(* IEC 61131-3 sources: BnR-PLC-motor-configuration/ncsdcctrl, 3 files *)

(* ---- ncsdcctrl.var ---- *)
VAR
	gAxis01_oSetPosOld : INT := 0;
	gAxis02_oSetPosOld : INT := 0;
	gAxis03_oSetPosOld : INT := 0;
END_VAR

(* ---- ncsdcctrlCyclic.st ---- *)
PROGRAM _CYCLIC

(* ### BEGIN gAxis01 ### *)

(* life counter emulation of digital inputs *)
      gAxis01_DiDoIf.iLifeCntReference := gAxis01_DiDoIf.iLifeCntReference + 1;
      gAxis01_DiDoIf.iLifeCntNegHwEnd  := gAxis01_DiDoIf.iLifeCntNegHwEnd  + 1;
      gAxis01_DiDoIf.iLifeCntPosHwEnd  := gAxis01_DiDoIf.iLifeCntPosHwEnd  + 1;

(* default function model of ACOPOSmicro: convert absolute steps to delta steps - overflow save delta calculation *)
      gAxis01_MotorStep0 := gAxis01_DrvIf.oSetPos - gAxis01_oSetPosOld;
      gAxis01_oSetPosOld := gAxis01_DrvIf.oSetPos;

(* ### END gAxis01 ### *)

(* ### BEGIN gAxis02 ### *)

(* life counter emulation of digital inputs *)
      gAxis02_DiDoIf.iLifeCntReference := gAxis02_DiDoIf.iLifeCntReference + 1;
      gAxis02_DiDoIf.iLifeCntNegHwEnd  := gAxis02_DiDoIf.iLifeCntNegHwEnd  + 1;
      gAxis02_DiDoIf.iLifeCntPosHwEnd  := gAxis02_DiDoIf.iLifeCntPosHwEnd  + 1;

(* default function model of ACOPOSmicro: convert absolute steps to delta steps - overflow save delta calculation *)
      gAxis02_MotorStep0 := gAxis02_DrvIf.oSetPos - gAxis02_oSetPosOld;
      gAxis02_oSetPosOld := gAxis02_DrvIf.oSetPos;

(* ### END gAxis02 ### *)

(* ### BEGIN gAxis03 ### *)

(* life counter emulation of digital inputs *)
      gAxis03_DiDoIf.iLifeCntReference := gAxis03_DiDoIf.iLifeCntReference + 1;
      gAxis03_DiDoIf.iLifeCntNegHwEnd  := gAxis03_DiDoIf.iLifeCntNegHwEnd  + 1;
      gAxis03_DiDoIf.iLifeCntPosHwEnd  := gAxis03_DiDoIf.iLifeCntPosHwEnd  + 1;

(* default function model of ACOPOSmicro: convert absolute steps to delta steps - overflow save delta calculation *)
      gAxis03_MotorStep0 := gAxis03_DrvIf.oSetPos - gAxis03_oSetPosOld;
      gAxis03_oSetPosOld := gAxis03_DrvIf.oSetPos;

(* ### END gAxis03 ### *)

END_PROGRAM

(* ---- ncsdcctrlInit.st ---- *)
PROGRAM _INIT

(* ### BEGIN gAxis01 ### *)

(* initialize general interfaces *)
      gAxis01.size := gAxis01.size;
      gAxis01_HW.DrvIf_Typ := ncSDC_DRVSM16;
      brsstrcpy( ADR(gAxis01_HW.DrvIf_Name[0]), ADR('gAxis01_DrvIf') );
      gAxis01_HW.DiDoIf_Typ := ncSDC_DIDO;
      brsstrcpy( ADR(gAxis01_HW.DiDoIf_Name[0]), ADR('gAxis01_DiDoIf') );
      gAxis01_HW.EncIf1_Typ := ncSDC_ENC16;
      brsstrcpy( ADR(gAxis01_HW.EncIf1_Name[0]), ADR('gAxis01_EncIf1') );
      gAxis01_EncIf1.iLifeCnt := gAxis01_EncIf1.iLifeCnt;

(* initialize old-value for delta step calculation *)
      gAxis01_oSetPosOld := gAxis01_DrvIf.oSetPos;

(* ### END gAxis01 ### *)

(* ### BEGIN gAxis02 ### *)

(* initialize general interfaces *)
      gAxis02.size := gAxis02.size;
      gAxis02_HW.DrvIf_Typ := ncSDC_DRVSM16;
      brsstrcpy( ADR(gAxis02_HW.DrvIf_Name[0]), ADR('gAxis02_DrvIf') );
      gAxis02_HW.DiDoIf_Typ := ncSDC_DIDO;
      brsstrcpy( ADR(gAxis02_HW.DiDoIf_Name[0]), ADR('gAxis02_DiDoIf') );
      gAxis02_HW.EncIf1_Typ := ncSDC_ENC16;
      brsstrcpy( ADR(gAxis02_HW.EncIf1_Name[0]), ADR('gAxis02_EncIf1') );
      gAxis02_EncIf1.iLifeCnt := gAxis02_EncIf1.iLifeCnt;

(* initialize old-value for delta step calculation *)
      gAxis02_oSetPosOld := gAxis02_DrvIf.oSetPos;

(* ### END gAxis02 ### *)

(* ### BEGIN gAxis03 ### *)

(* initialize general interfaces *)
      gAxis03.size := gAxis03.size;
      gAxis03_HW.DrvIf_Typ := ncSDC_DRVSM16;
      brsstrcpy( ADR(gAxis03_HW.DrvIf_Name[0]), ADR('gAxis03_DrvIf') );
      gAxis03_HW.DiDoIf_Typ := ncSDC_DIDO;
      brsstrcpy( ADR(gAxis03_HW.DiDoIf_Name[0]), ADR('gAxis03_DiDoIf') );
      gAxis03_HW.EncIf1_Typ := ncSDC_ENC16;
      brsstrcpy( ADR(gAxis03_HW.EncIf1_Name[0]), ADR('gAxis03_EncIf1') );
      gAxis03_EncIf1.iLifeCnt := gAxis03_EncIf1.iLifeCnt;

(* initialize old-value for delta step calculation *)
      gAxis03_oSetPosOld := gAxis03_DrvIf.oSetPos;

(* ### END gAxis03 ### *)

END_PROGRAM
